TYPE ST_SettingsPalletConveyor :
STRUCT
	rSpeedManual : LREAL := 50.0; //Speed for manual control [default: 50.0 mm/s]
	rSpeedGoToCentering : LREAL := 100.0; //Speed to move to centering position [default: 100.0 mm/s]
	rSpeedGoToDocking : LREAL := 50.0; //Speed to move to docking position [default: 50.0 mm/s]
	rSpeedReturnToInfeed : LREAL := 100.0; //Speed to move (back) to infeed position [default: 100.0 mm/s]
END_STRUCT
END_TYPE

(* stored: Version 1.1.0.1, ProductVersion 3.1.4024.12
   DUT ST_SettingsPalletConveyor: Id {17185faa-8192-4589-aff2-b3f618a709c5} *)
